// TwinCAT 3 PLC project PLC
// Company: Test
// ProjectVersion: 1.1.10
// ProgramVersion: 3.1.4026.1+972e9c44872ad038b353624a861fd7e3244e9f75
// libraries:
//   Tc2_Standard, * (Beckhoff Automation GmbH)
//   Tc2_System, * (Beckhoff Automation GmbH)
// project tree:
//   / PlcTask.TcTTO
//   POUs/ MAIN.TcPOU
// real-time tasks:
//   TASK PlcTask: cycle T#10ms, priority 20, ADS port 350

CONFIGURATION PLC
    RESOURCE PLC ON TwinCAT3
        TASK PlcTask(INTERVAL := T#10ms, PRIORITY := 20);
        PROGRAM MAIN WITH PlcTask : MAIN;
    END_RESOURCE
END_CONFIGURATION

// ---- POUs/MAIN.TcPOU
PROGRAM MAIN
VAR
	{ attribute 'TcHmiSymbol.AddSymbol' }
	nCtx			: DINT;
	
	{ attribute 'My.Custom.Attribute' := 'Attribute value' }
	{ attribute 'TcHmiSymbol.AddSymbol' }
	nAttribute		: DINT;
	ton				: TON;
END_VAR

ton(IN:=NOT ton.Q, PT:=T#5S);
IF ton.Q THEN
	nAttribute := nAttribute + 1;
END_IF

END_PROGRAM
